TYPE ST_EL70xx_POS_Status :
STRUCT
	Busy  			AT%I* : BIT;
	InTarget  		AT%I* : BIT;
	Warning  		AT%I* : BIT;
	Error 			AT%I* : BIT;
	Calibrated  	AT%I* : BIT;
	//ReadyToExecute  AT%I* : BIT;
	ActualPosition  AT%I* : DINT;
END_STRUCT
END_TYPE

(* stored: Version 1.1.0.1, ProductVersion 3.1.4024.11
   DUT ST_EL70xx_POS_Status: Id {4f52ecb2-1c87-43b4-9584-030ec6e0cd11} *)
